FUNCTION_BLOCK FB_RedColor IMPLEMENTS ITF_Color

METHOD applyColor : STRING
applyColor := 'red';
END_METHOD

END_FUNCTION_BLOCK

(* stored: Version 1.1.0.1, ProductVersion 3.1.4024.12
   POU FB_RedColor: Id {e01cb8a2-a3a4-4ebd-ae69-49d31664ab7c}, SpecialFunc None
   Method applyColor: Id {357c017a-3121-4992-af3f-056bb7babd1e} *)
